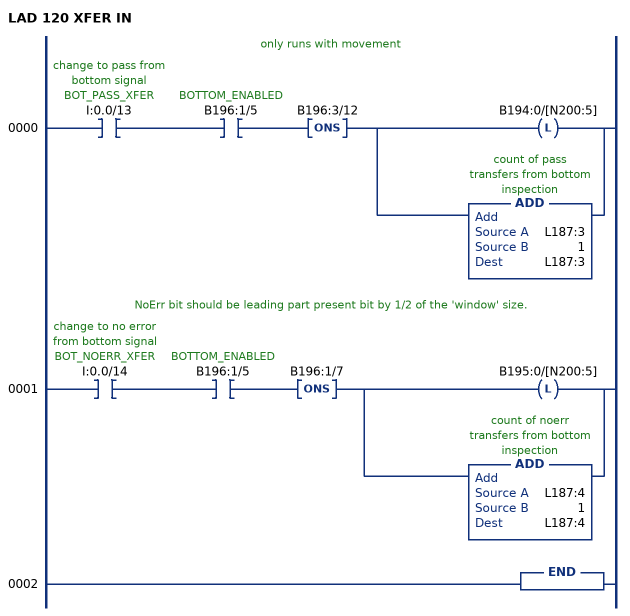
% Rung: 0 %
% only runs with movement %
SOR XIC I:0.0/13 XIC B196:1/5 ONS B196:3/12 BST OTL B194:0/[N200:5] NXB ADD L187:3 1 L187:3 BND EOR
%   I:0.0/13  BOT_PASS_XFER  "change to pass from bottom signal" %
%   B196:1/5  BOTTOM_ENABLED %
%   N200:5  TOP_LOAD %
%   L187:3  "count of pass transfers from bottom inspection" %
% Rung: 1 %
% NoErr bit should be leading part present bit by 1/2 of the 'window' size. %
SOR XIC I:0.0/14 XIC B196:1/5 ONS B196:1/7 BST OTL B195:0/[N200:5] NXB ADD L187:4 1 L187:4 BND EOR
%   I:0.0/14  BOT_NOERR_XFER  "change to no error from bottom signal" %
%   B196:1/5  BOTTOM_ENABLED %
%   N200:5  TOP_LOAD %
%   L187:4  "count of noerr transfers from bottom inspection" %
% Rung: 2 %
SOR END EOR

LADDER 121 "SIM PARTS"
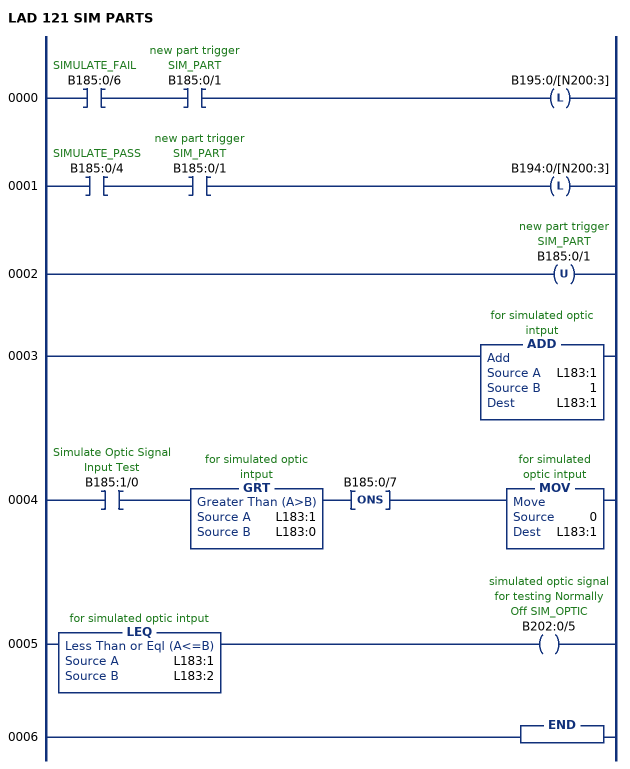
% Rung: 0 %
SOR XIC B185:0/6 XIC B185:0/1 OTL B195:0/[N200:3] EOR
%   B185:0/6  SIMULATE_FAIL %
%   B185:0/1  SIM_PART  "new part trigger" %
%   N200:3  OPT_LD_PT %
% Rung: 1 %
SOR XIC B185:0/4 XIC B185:0/1 OTL B194:0/[N200:3] EOR
%   B185:0/4  SIMULATE_PASS %
%   B185:0/1  SIM_PART  "new part trigger" %
%   N200:3  OPT_LD_PT %
% Rung: 2 %
SOR OTU B185:0/1 EOR
%   B185:0/1  SIM_PART  "new part trigger" %
% Rung: 3 %
SOR ADD L183:1 1 L183:1 EOR
%   L183:1  "for simulated optic intput" %
% Rung: 4 %
SOR XIC B185:1/0 GRT L183:1 L183:0 ONS B185:0/7 MOV 0 L183:1 EOR
%   B185:1/0  "Simulate Optic Signal Input Test" %
%   L183:1  "for simulated optic intput" %
%   L183:0  "Movement pulse count for part data injection" %
% Rung: 5 %
SOR LEQ L183:1 L183:2 OTE B202:0/5 EOR
%   L183:1  "for simulated optic intput" %
%   L183:2  "simulated part width" %
%   B202:0/5  SIM_OPTIC  "simulated optic signal for testing Normally Off" %
% Rung: 6 %
SOR END EOR

LADDER 122 "PARTDETECT"
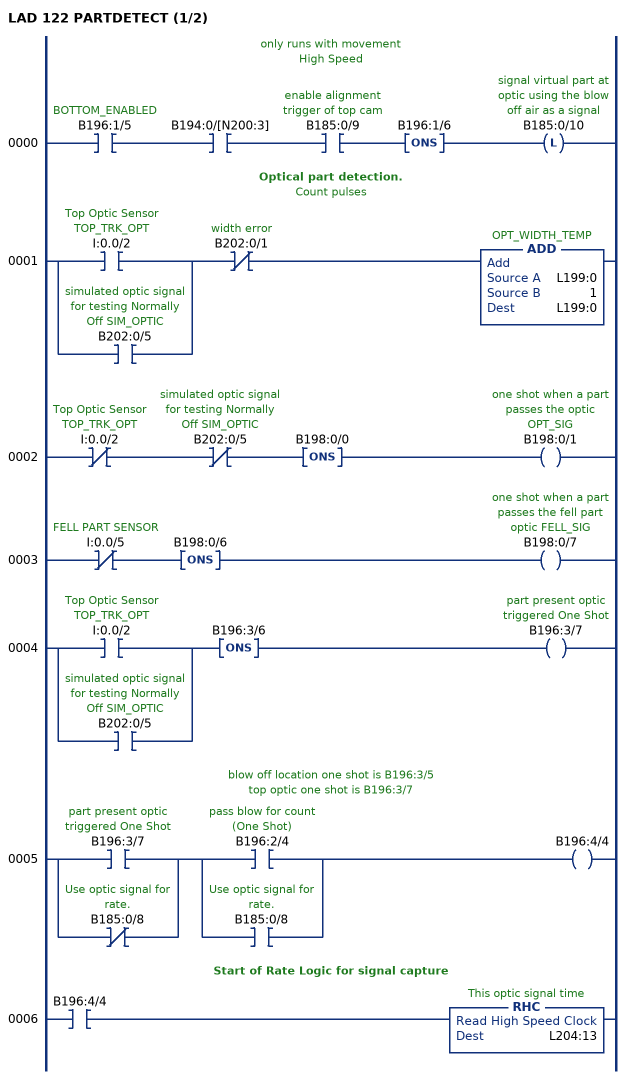
% Rung: 0 %
% only runs with movement
% High Speed %
SOR XIC B196:1/5 XIC B194:0/[N200:3] XIC B185:0/9 ONS B196:1/6 OTL B185:0/10 EOR
%   B196:1/5  BOTTOM_ENABLED %
%   N200:3  OPT_LD_PT %
%   B185:0/9  "enable alignment trigger of top cam" %
%   B185:0/10  "signal virtual part at optic using the blow off air as a signal" %
% Rung: 1 %
% TITLE: Optical part detection. %
% Count pulses %
SOR BST XIC I:0.0/2 NXB XIC B202:0/5 BND XIO B202:0/1 ADD L199:0 1 L199:0 EOR
%   I:0.0/2  TOP_TRK_OPT  "Top Optic Sensor" %
%   B202:0/5  SIM_OPTIC  "simulated optic signal for testing Normally Off" %
%   B202:0/1  "width error" %
%   L199:0  OPT_WIDTH_TEMP %
% Rung: 2 %
SOR XIO I:0.0/2 XIO B202:0/5 ONS B198:0/0 OTE B198:0/1 EOR
%   I:0.0/2  TOP_TRK_OPT  "Top Optic Sensor" %
%   B202:0/5  SIM_OPTIC  "simulated optic signal for testing Normally Off" %
%   B198:0/1  OPT_SIG  "one shot when a part passes the optic" %
% Rung: 3 %
SOR XIO I:0.0/5 ONS B198:0/6 OTE B198:0/7 EOR
%   I:0.0/5  "FELL PART SENSOR" %
%   B198:0/7  FELL_SIG  "one shot when a part passes the fell part optic" %
% Rung: 4 %
SOR BST XIC I:0.0/2 NXB XIC B202:0/5 BND ONS B196:3/6 OTE B196:3/7 EOR
%   I:0.0/2  TOP_TRK_OPT  "Top Optic Sensor" %
%   B202:0/5  SIM_OPTIC  "simulated optic signal for testing Normally Off" %
%   B196:3/7  "part present optic triggered One Shot" %
% Rung: 5 %
% blow off location one shot is B196:3/5
% top optic one shot is B196:3/7 %
SOR BST XIC B196:3/7 NXB XIO B185:0/8 BND BST XIC B196:2/4 NXB XIC B185:0/8 BND OTE B196:4/4 EOR
%   B196:3/7  "part present optic triggered One Shot" %
%   B185:0/8  "Use optic signal for rate." %
%   B196:2/4  "pass blow for count (One Shot)" %
% Rung: 6 %
% TITLE: Start of Rate Logic for signal capture %
SOR XIC B196:4/4 RHC L204:13 EOR
%   L204:13  "This optic signal time" %

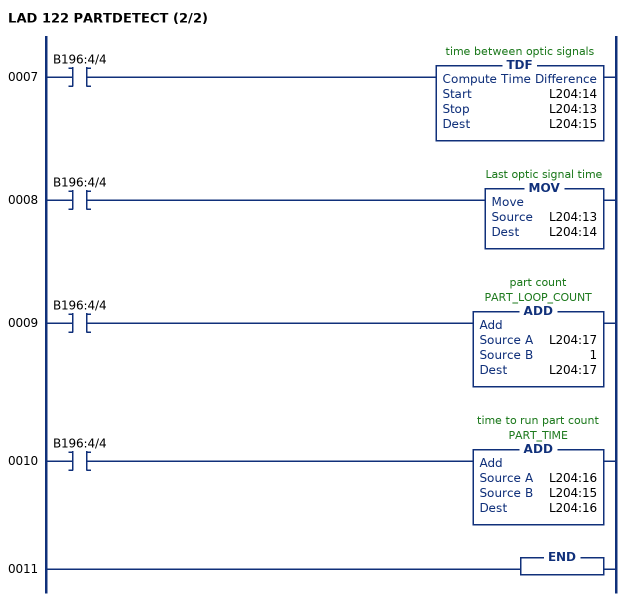
% Rung: 7 %
SOR XIC B196:4/4 TDF L204:14 L204:13 L204:15 EOR
%   L204:14  "Last optic signal time" %
%   L204:13  "This optic signal time" %
%   L204:15  "time between optic signals" %
% Rung: 8 %
SOR XIC B196:4/4 MOV L204:13 L204:14 EOR
%   L204:13  "This optic signal time" %
%   L204:14  "Last optic signal time" %
% Rung: 9 %
SOR XIC B196:4/4 ADD L204:17 1 L204:17 EOR
%   L204:17  PART_LOOP_COUNT  "part count" %
% Rung: 10 %
SOR XIC B196:4/4 ADD L204:16 L204:15 L204:16 EOR
%   L204:16  PART_TIME  "time to run part count" %
%   L204:15  "time between optic signals" %
% Rung: 11 %
SOR END EOR

LADDER 123 "OPTICWIDTH"
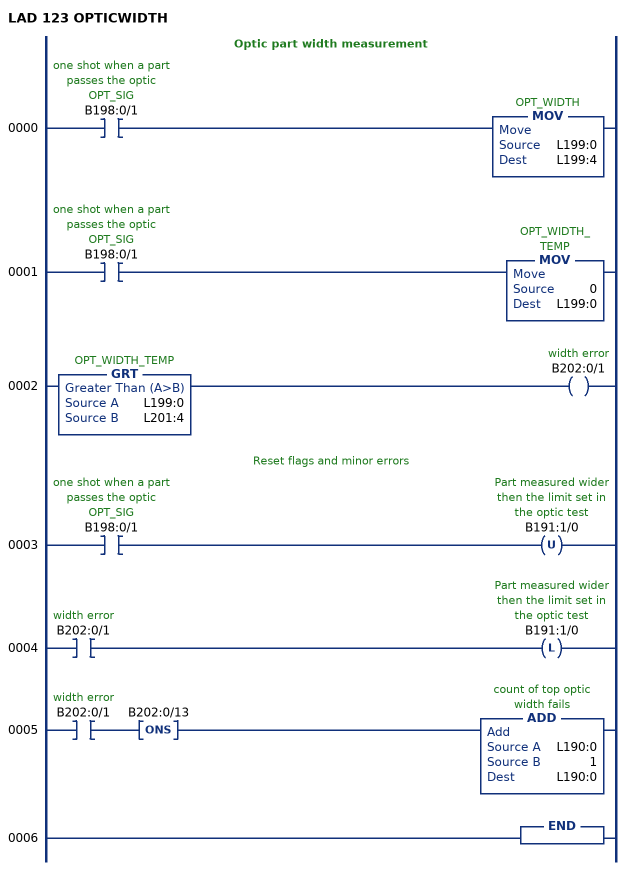
% Rung: 0 %
% TITLE: Optic part width measurement %
SOR XIC B198:0/1 MOV L199:0 L199:4 EOR
%   B198:0/1  OPT_SIG  "one shot when a part passes the optic" %
%   L199:0  OPT_WIDTH_TEMP %
%   L199:4  OPT_WIDTH %
% Rung: 1 %
SOR XIC B198:0/1 MOV 0 L199:0 EOR
%   B198:0/1  OPT_SIG  "one shot when a part passes the optic" %
%   L199:0  OPT_WIDTH_TEMP %
% Rung: 2 %
SOR GRT L199:0 L201:4 OTE B202:0/1 EOR
%   L199:0  OPT_WIDTH_TEMP %
%   L201:4  MAX_WIDTH  "hmi in" %
%   B202:0/1  "width error" %
% Rung: 3 %
% Reset flags and minor errors %
SOR XIC B198:0/1 OTU B191:1/0 EOR
%   B198:0/1  OPT_SIG  "one shot when a part passes the optic" %
%   B191:1/0  "Part measured wider then the limit set in the optic test" %
% Rung: 4 %
SOR XIC B202:0/1 OTL B191:1/0 EOR
%   B202:0/1  "width error" %
%   B191:1/0  "Part measured wider then the limit set in the optic test" %
% Rung: 5 %
SOR XIC B202:0/1 ONS B202:0/13 ADD L190:0 1 L190:0 EOR
%   B202:0/1  "width error" %
%   L190:0  "count of top optic width fails" %
% Rung: 6 %
SOR END EOR

LADDER 124 "PART GAP"
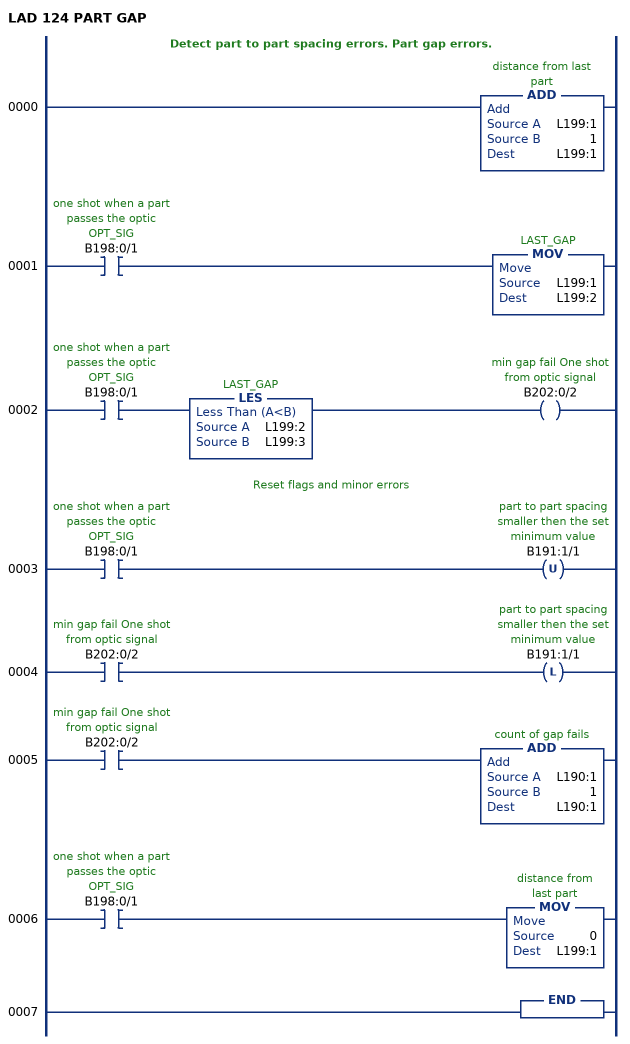
% Rung: 0 %
% TITLE: Detect part to part spacing errors. Part gap errors. %
SOR ADD L199:1 1 L199:1 EOR
%   L199:1  "distance from last part" %
% Rung: 1 %
SOR XIC B198:0/1 MOV L199:1 L199:2 EOR
%   B198:0/1  OPT_SIG  "one shot when a part passes the optic" %
%   L199:1  "distance from last part" %
%   L199:2  LAST_GAP %
% Rung: 2 %
SOR XIC B198:0/1 LES L199:2 L199:3 OTE B202:0/2 EOR
%   B198:0/1  OPT_SIG  "one shot when a part passes the optic" %
%   L199:2  LAST_GAP %
%   L199:3  MIN_WIDTH %
%   B202:0/2  "min gap fail One shot from optic signal" %
% Rung: 3 %
% Reset flags and minor errors %
SOR XIC B198:0/1 OTU B191:1/1 EOR
%   B198:0/1  OPT_SIG  "one shot when a part passes the optic" %
%   B191:1/1  "part to part spacing smaller then the set minimum value" %
% Rung: 4 %
SOR XIC B202:0/2 OTL B191:1/1 EOR
%   B202:0/2  "min gap fail One shot from optic signal" %
%   B191:1/1  "part to part spacing smaller then the set minimum value" %
% Rung: 5 %
SOR XIC B202:0/2 ADD L190:1 1 L190:1 EOR
%   B202:0/2  "min gap fail One shot from optic signal" %
%   L190:1  "count of gap fails" %
% Rung: 6 %
SOR XIC B198:0/1 MOV 0 L199:1 EOR
%   B198:0/1  OPT_SIG  "one shot when a part passes the optic" %
%   L199:1  "distance from last part" %
% Rung: 7 %
SOR END EOR

LADDER 125 "OPTIC CL"
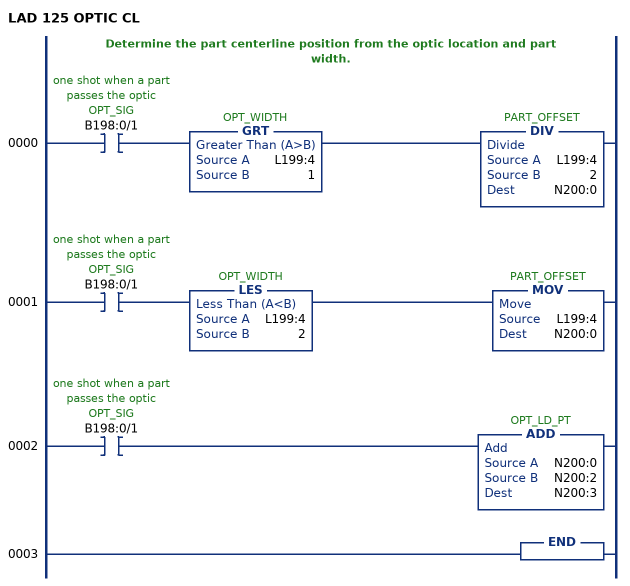
% Rung: 0 %
% TITLE: Determine the part centerline position from the optic location and part width. %
SOR XIC B198:0/1 GRT L199:4 1 DIV L199:4 2 N200:0 EOR
%   B198:0/1  OPT_SIG  "one shot when a part passes the optic" %
%   L199:4  OPT_WIDTH %
%   N200:0  PART_OFFSET %
% Rung: 1 %
SOR XIC B198:0/1 LES L199:4 2 MOV L199:4 N200:0 EOR
%   B198:0/1  OPT_SIG  "one shot when a part passes the optic" %
%   L199:4  OPT_WIDTH %
%   N200:0  PART_OFFSET %
% Rung: 2 %
SOR XIC B198:0/1 ADD N200:0 N200:2 N200:3 EOR
%   B198:0/1  OPT_SIG  "one shot when a part passes the optic" %
%   N200:0  PART_OFFSET %
%   N200:2  OPTIC_LOC %
%   N200:3  OPT_LD_PT %
% Rung: 3 %
SOR END EOR

LADDER 126 "ALIGNMENT"
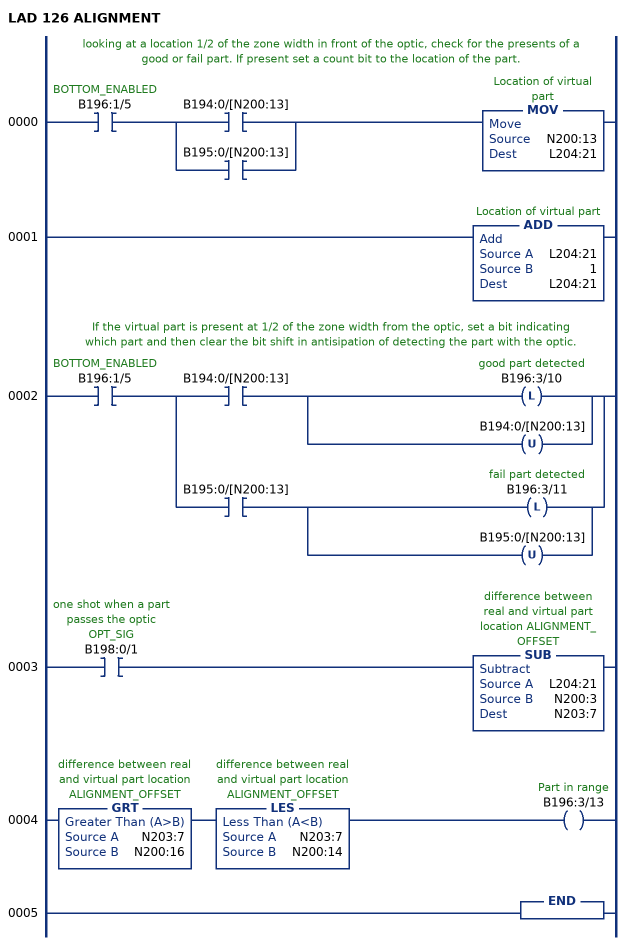
% Rung: 0 %
% looking at a location 1/2 of the zone width in front of the optic, check for the presents of a good or fail part. If present set a count bit to the location of the part. %
SOR XIC B196:1/5 BST XIC B194:0/[N200:13] NXB XIC B195:0/[N200:13] BND MOV N200:13 L204:21 EOR
%   B196:1/5  BOTTOM_ENABLED %
%   N200:13  ALIGNMENT_START_LOC %
%   L204:21  "Location of virtual part" %
% Rung: 1 %
SOR ADD L204:21 1 L204:21 EOR
%   L204:21  "Location of virtual part" %
% Rung: 2 %
% If the virtual part is present at 1/2 of the zone width from the optic, set a bit indicating which part and then clear the bit shift in antisipation of detecting the part with the optic. %
SOR XIC B196:1/5 BST XIC B194:0/[N200:13] BST OTL B196:3/10 NXB OTU B194:0/[N200:13] BND NXB XIC B195:0/[N200:13] BST OTL B196:3/11 NXB OTU B195:0/[N200:13] BND BND EOR
%   B196:1/5  BOTTOM_ENABLED %
%   N200:13  ALIGNMENT_START_LOC %
%   B196:3/10  "good part detected" %
%   B196:3/11  "fail part detected" %
% Rung: 3 %
SOR XIC B198:0/1 SUB L204:21 N200:3 N203:7 EOR
%   B198:0/1  OPT_SIG  "one shot when a part passes the optic" %
%   L204:21  "Location of virtual part" %
%   N200:3  OPT_LD_PT %
%   N203:7  ALIGNMENT_OFFSET  "difference between real and virtual part location" %
% Rung: 4 %
SOR GRT N203:7 N200:16 LES N203:7 N200:14 OTE B196:3/13 EOR
%   N203:7  ALIGNMENT_OFFSET  "difference between real and virtual part location" %
%   N200:16  "Minus one half of the transition zone" %
%   N200:14  "1/2 transistion zone" %
%   B196:3/13  "Part in range" %
% Rung: 5 %
SOR END EOR

LADDER 127 "OPTIC_LOAD"
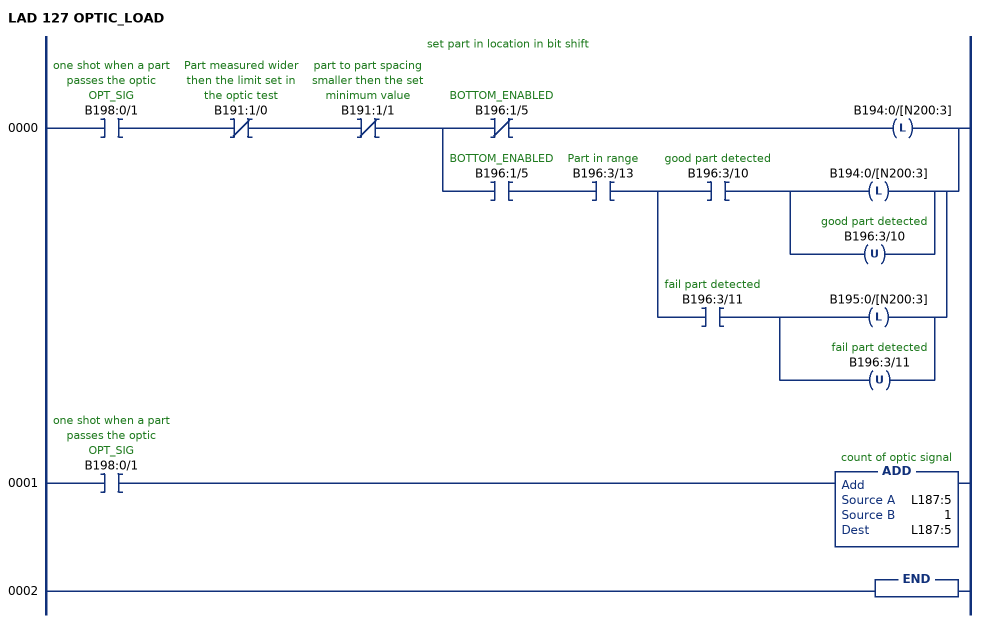
% Rung: 0 %
% set part in location in bit shift %
SOR XIC B198:0/1 XIO B191:1/0 XIO B191:1/1 BST XIO B196:1/5 OTL B194:0/[N200:3] NXB XIC B196:1/5 XIC B196:3/13 BST XIC B196:3/10 BST OTL B194:0/[N200:3] NXB OTU B196:3/10 BND NXB XIC B196:3/11 BST OTL B195:0/[N200:3] NXB OTU B196:3/11 BND BND BND EOR
%   B198:0/1  OPT_SIG  "one shot when a part passes the optic" %
%   B191:1/0  "Part measured wider then the limit set in the optic test" %
%   B191:1/1  "part to part spacing smaller then the set minimum value" %
%   B196:1/5  BOTTOM_ENABLED %
%   N200:3  OPT_LD_PT %
%   B196:3/13  "Part in range" %
%   B196:3/10  "good part detected" %
%   B196:3/11  "fail part detected" %
% Rung: 1 %
SOR XIC B198:0/1 ADD L187:5 1 L187:5 EOR
%   B198:0/1  OPT_SIG  "one shot when a part passes the optic" %
%   L187:5  "count of optic signal" %
% Rung: 2 %
SOR END EOR

LADDER 128 "FELL PART"
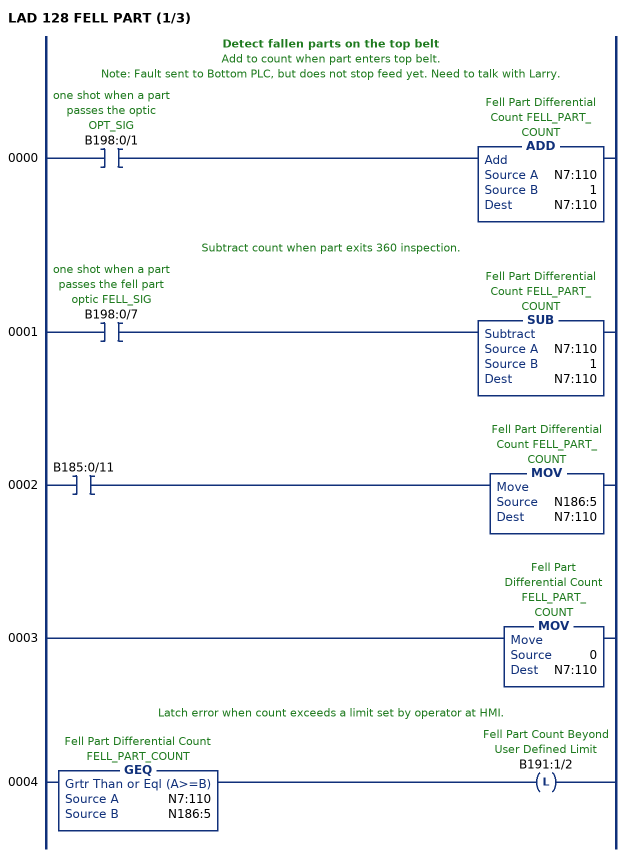
% Rung: 0 %
% TITLE: Detect fallen parts on the top belt %
% Add to count when part enters top belt.
% Note: Fault sent to Bottom PLC, but does not stop feed yet. Need to talk with Larry. %
SOR XIC B198:0/1 ADD N7:110 1 N7:110 EOR
%   B198:0/1  OPT_SIG  "one shot when a part passes the optic" %
%   N7:110  FELL_PART_COUNT  "Fell Part Differential Count" %
% Rung: 1 %
% Subtract count when part exits 360 inspection. %
SOR XIC B198:0/7 SUB N7:110 1 N7:110 EOR
%   B198:0/7  FELL_SIG  "one shot when a part passes the fell part optic" %
%   N7:110  FELL_PART_COUNT  "Fell Part Differential Count" %
% Rung: 2 %
SOR XIC B185:0/11 MOV N186:5 N7:110 EOR
%   N186:5  FELL_PART_LIMIT  "Fell Part Differential Limit From HMI" %
%   N7:110  FELL_PART_COUNT  "Fell Part Differential Count" %
% Rung: 3 %
SOR MOV 0 N7:110 EOR
%   N7:110  FELL_PART_COUNT  "Fell Part Differential Count" %
% Rung: 4 %
% Latch error when count exceeds a limit set by operator at HMI. %
SOR GEQ N7:110 N186:5 OTL B191:1/2 EOR
%   N7:110  FELL_PART_COUNT  "Fell Part Differential Count" %
%   N186:5  FELL_PART_LIMIT  "Fell Part Differential Limit From HMI" %
%   B191:1/2  "Fell Part Count Beyond User Defined Limit" %

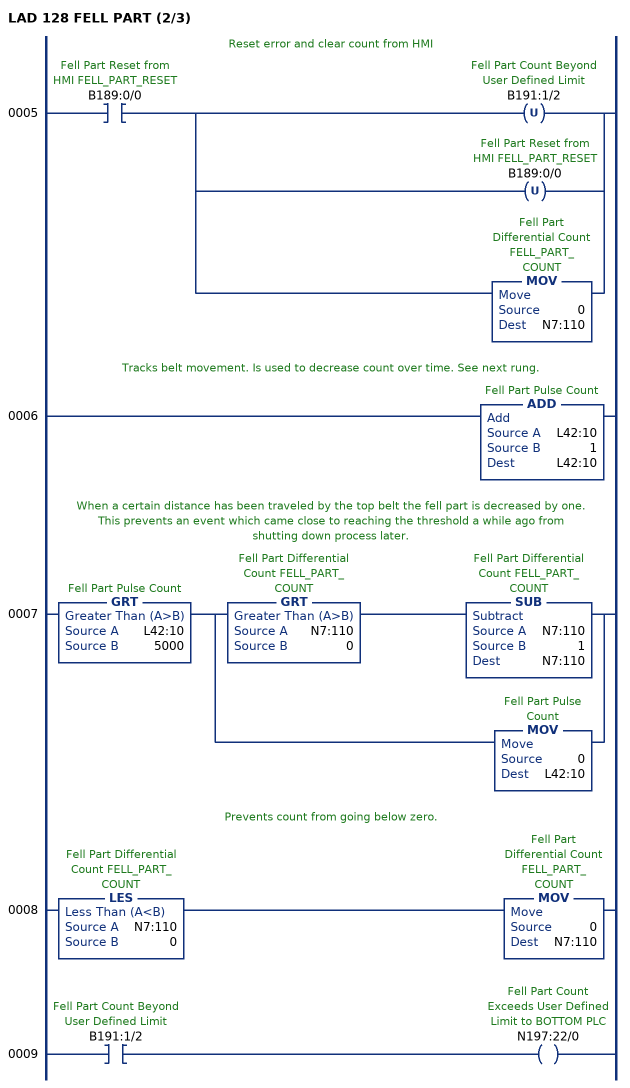
% Rung: 5 %
% Reset error and clear count from HMI %
SOR XIC B189:0/0 BST OTU B191:1/2 NXB OTU B189:0/0 NXB MOV 0 N7:110 BND EOR
%   B189:0/0  FELL_PART_RESET  "Fell Part Reset from HMI" %
%   B191:1/2  "Fell Part Count Beyond User Defined Limit" %
%   N7:110  FELL_PART_COUNT  "Fell Part Differential Count" %
% Rung: 6 %
% Tracks belt movement. Is used to decrease count over time. See next rung. %
SOR ADD L42:10 1 L42:10 EOR
%   L42:10  "Fell Part Pulse Count" %
% Rung: 7 %
% When a certain distance has been traveled by the top belt the fell part is decreased by one. This prevents an event which came close to reaching the threshold a while ago from shutting down process later. %
SOR GRT L42:10 5000 BST GRT N7:110 0 SUB N7:110 1 N7:110 NXB MOV 0 L42:10 BND EOR
%   L42:10  "Fell Part Pulse Count" %
%   N7:110  FELL_PART_COUNT  "Fell Part Differential Count" %
% Rung: 8 %
% Prevents count from going below zero. %
SOR LES N7:110 0 MOV 0 N7:110 EOR
%   N7:110  FELL_PART_COUNT  "Fell Part Differential Count" %
% Rung: 9 %
SOR XIC B191:1/2 OTE N197:22/0 EOR
%   B191:1/2  "Fell Part Count Beyond User Defined Limit" %
%   N197:22/0  "Fell Part Count Exceeds User Defined Limit to BOTTOM PLC" %

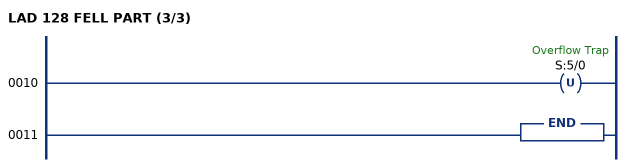
% Rung: 10 %
SOR OTU S:5/0 EOR
%   S:5/0  "Overflow Trap" %
% Rung: 11 %
SOR END EOR

LADDER 130 "INS 5 TRIG"
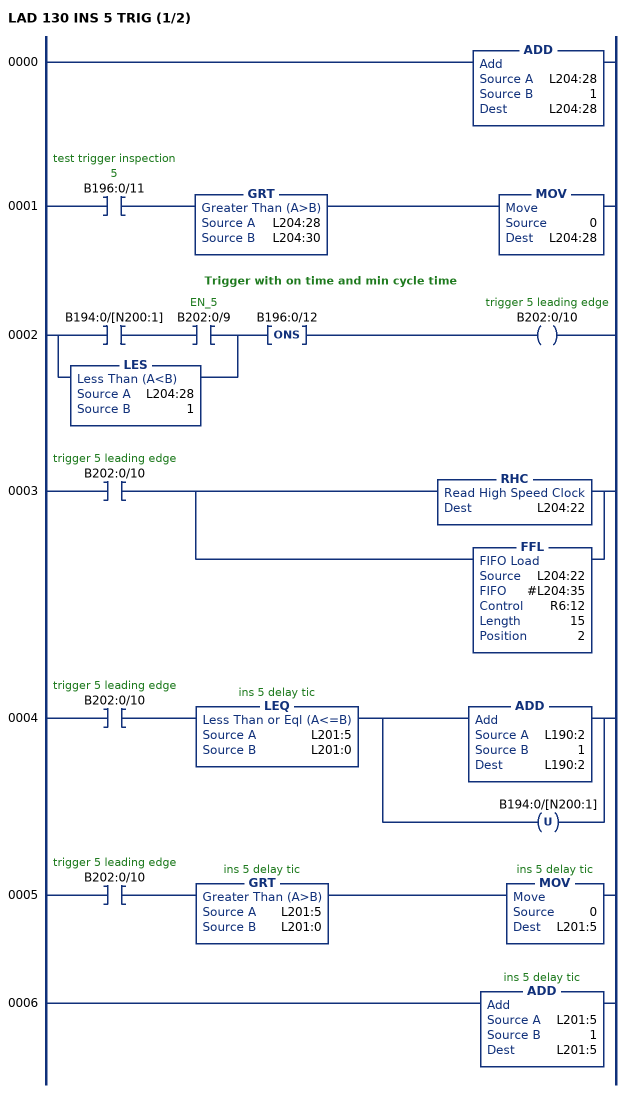
% Rung: 0 %
SOR ADD L204:28 1 L204:28 EOR
% Rung: 1 %
SOR XIC B196:0/11 GRT L204:28 L204:30 MOV 0 L204:28 EOR
%   B196:0/11  "test trigger inspection 5" %
% Rung: 2 %
% TITLE: Trigger with on time and min cycle time %
SOR BST XIC B194:0/[N200:1] XIC B202:0/9 NXB LES L204:28 1 BND ONS B196:0/12 OTE B202:0/10 EOR
%   N200:1  INS_5_TRIG_LOC %
%   B202:0/9  EN_5 %
%   B202:0/10  "trigger 5 leading edge" %
% Rung: 3 %
SOR XIC B202:0/10 BST RHC L204:22 NXB FFL L204:22 #L204:35 R6:12 15 2 BND EOR
%   B202:0/10  "trigger 5 leading edge" %
% Rung: 4 %
SOR XIC B202:0/10 LEQ L201:5 L201:0 BST ADD L190:2 1 L190:2 NXB OTU B194:0/[N200:1] BND EOR
%   B202:0/10  "trigger 5 leading edge" %
%   L201:5  "ins 5 delay tic" %
%   L201:0  CAM_5_MIN_CYCLE_TIME %
%   N200:1  INS_5_TRIG_LOC %
% Rung: 5 %
SOR XIC B202:0/10 GRT L201:5 L201:0 MOV 0 L201:5 EOR
%   B202:0/10  "trigger 5 leading edge" %
%   L201:5  "ins 5 delay tic" %
%   L201:0  CAM_5_MIN_CYCLE_TIME %
% Rung: 6 %
SOR ADD L201:5 1 L201:5 EOR
%   L201:5  "ins 5 delay tic" %

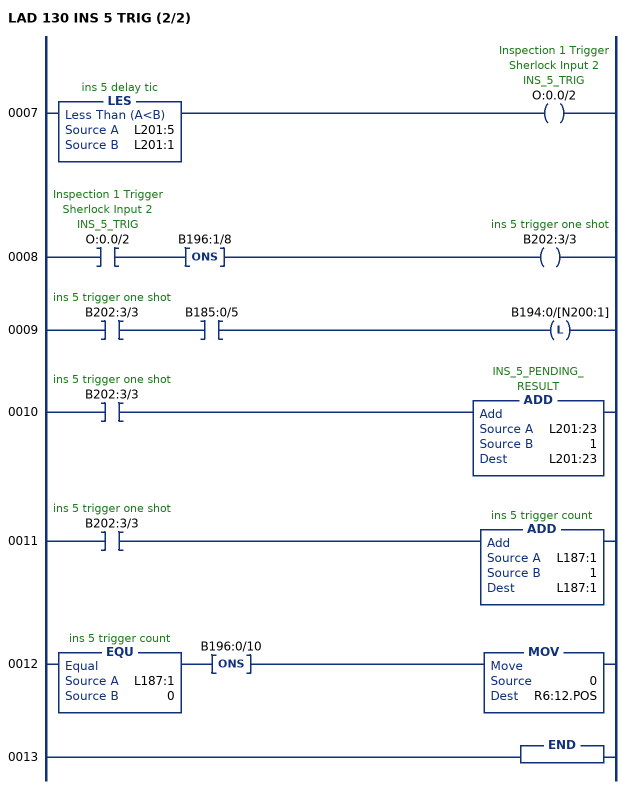
% Rung: 7 %
SOR LES L201:5 L201:1 OTE O:0.0/2 EOR
%   L201:5  "ins 5 delay tic" %
%   L201:1  CAM_5_TRIG_TIME %
%   O:0.0/2  INS_5_TRIG  "Inspection 1 Trigger Sherlock Input 2" %
% Rung: 8 %
SOR XIC O:0.0/2 ONS B196:1/8 OTE B202:3/3 EOR
%   O:0.0/2  INS_5_TRIG  "Inspection 1 Trigger Sherlock Input 2" %
%   B202:3/3  "ins 5 trigger one shot" %
% Rung: 9 %
SOR XIC B202:3/3 XIC B185:0/5 OTL B194:0/[N200:1] EOR
%   B202:3/3  "ins 5 trigger one shot" %
%   N200:1  INS_5_TRIG_LOC %
% Rung: 10 %
SOR XIC B202:3/3 ADD L201:23 1 L201:23 EOR
%   B202:3/3  "ins 5 trigger one shot" %
%   L201:23  INS_5_PENDING_RESULT %
% Rung: 11 %
SOR XIC B202:3/3 ADD L187:1 1 L187:1 EOR
%   B202:3/3  "ins 5 trigger one shot" %
%   L187:1  "ins 5 trigger count" %
% Rung: 12 %
SOR EQU L187:1 0 ONS B196:0/10 MOV 0 R6:12.POS EOR
%   L187:1  "ins 5 trigger count" %
% Rung: 13 %
SOR END EOR

LADDER 131 "INS 5 RSLT"
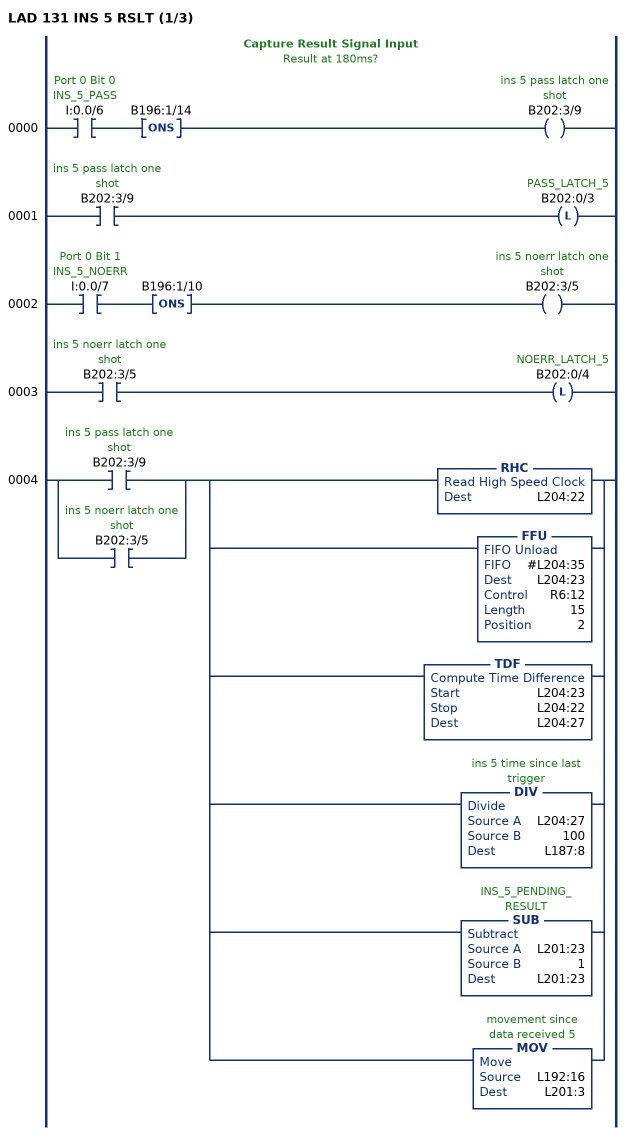
% Rung: 0 %
% TITLE: Capture Result Signal Input %
% Result at 180ms? %
SOR XIC I:0.0/6 ONS B196:1/14 OTE B202:3/9 EOR
%   I:0.0/6  INS_5_PASS  "Port 0 Bit 0" %
%   B202:3/9  "ins 5 pass latch one shot" %
% Rung: 1 %
SOR XIC B202:3/9 OTL B202:0/3 EOR
%   B202:3/9  "ins 5 pass latch one shot" %
%   B202:0/3  PASS_LATCH_5 %
% Rung: 2 %
SOR XIC I:0.0/7 ONS B196:1/10 OTE B202:3/5 EOR
%   I:0.0/7  INS_5_NOERR  "Port 0 Bit 1" %
%   B202:3/5  "ins 5 noerr latch one shot" %
% Rung: 3 %
SOR XIC B202:3/5 OTL B202:0/4 EOR
%   B202:3/5  "ins 5 noerr latch one shot" %
%   B202:0/4  NOERR_LATCH_5 %
% Rung: 4 %
SOR BST XIC B202:3/9 NXB XIC B202:3/5 BND BST RHC L204:22 NXB FFU #L204:35 L204:23 R6:12 15 2 NXB TDF L204:23 L204:22 L204:27 NXB DIV L204:27 100 L187:8 NXB SUB L201:23 1 L201:23 NXB MOV L192:16 L201:3 BND EOR
%   B202:3/9  "ins 5 pass latch one shot" %
%   B202:3/5  "ins 5 noerr latch one shot" %
%   L187:8  "ins 5 time since last trigger" %
%   L201:23  INS_5_PENDING_RESULT %
%   L192:16  COMBINED_OFFSET  "use this offset value for looking for the part present bit after an inspeciton" %
%   L201:3  "movement since data received 5" %

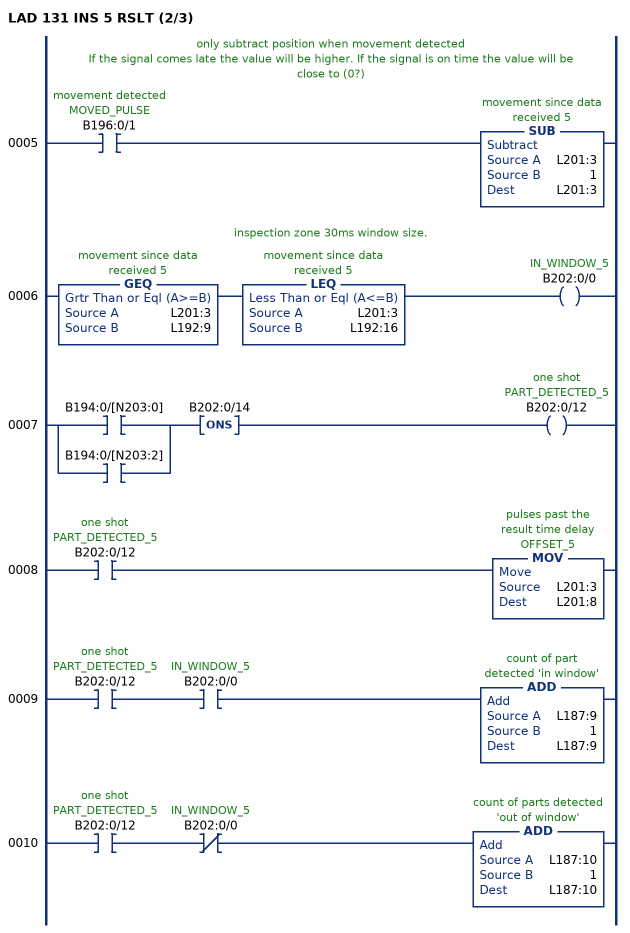
% Rung: 5 %
% only subtract position when movement detected
% If the signal comes late the value will be higher. If the signal is on time the value will be close to (0?) %
SOR XIC B196:0/1 SUB L201:3 1 L201:3 EOR
%   B196:0/1  MOVED_PULSE  "movement detected" %
%   L201:3  "movement since data received 5" %
% Rung: 6 %
% inspection zone 30ms window size. %
SOR GEQ L201:3 L192:9 LEQ L201:3 L192:16 OTE B202:0/0 EOR
%   L201:3  "movement since data received 5" %
%   L192:9  RESULT_OFFSET  "in pulses" %
%   L192:16  COMBINED_OFFSET  "use this offset value for looking for the part present bit after an inspeciton" %
%   B202:0/0  IN_WINDOW_5 %
% Rung: 7 %
SOR BST XIC B194:0/[N203:0] NXB XIC B194:0/[N203:2] BND ONS B202:0/14 OTE B202:0/12 EOR
%   N203:0  INS_5_TEST_LOC1  "result + offset shift" %
%   N203:2  INS_5_TEST_LOC2 %
%   B202:0/12  PART_DETECTED_5  "one shot" %
% Rung: 8 %
SOR XIC B202:0/12 MOV L201:3 L201:8 EOR
%   B202:0/12  PART_DETECTED_5  "one shot" %
%   L201:3  "movement since data received 5" %
%   L201:8  OFFSET_5  "pulses past the result time delay" %
% Rung: 9 %
SOR XIC B202:0/12 XIC B202:0/0 ADD L187:9 1 L187:9 EOR
%   B202:0/12  PART_DETECTED_5  "one shot" %
%   B202:0/0  IN_WINDOW_5 %
%   L187:9  "count of part detected 'in window'" %
% Rung: 10 %
SOR XIC B202:0/12 XIO B202:0/0 ADD L187:10 1 L187:10 EOR
%   B202:0/12  PART_DETECTED_5  "one shot" %
%   B202:0/0  IN_WINDOW_5 %
%   L187:10  "count of parts detected 'out of window'" %

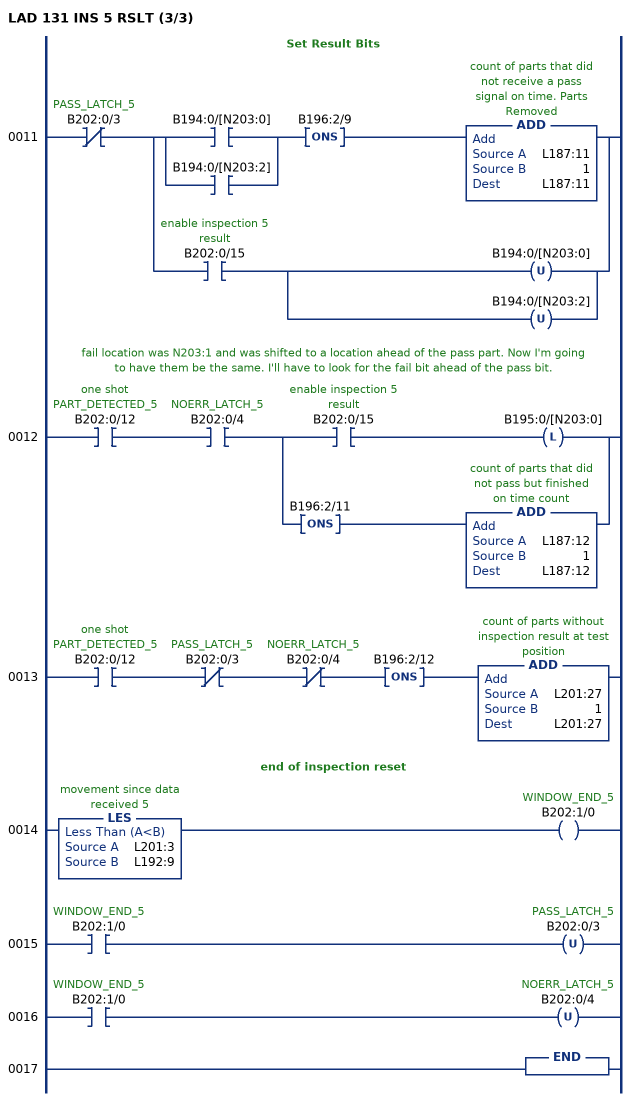
% Rung: 11 %
% TITLE: Set Result Bits %
SOR XIO B202:0/3 BST BST XIC B194:0/[N203:0] NXB XIC B194:0/[N203:2] BND ONS B196:2/9 ADD L187:11 1 L187:11 NXB XIC B202:0/15 BST OTU B194:0/[N203:0] NXB OTU B194:0/[N203:2] BND BND EOR
%   B202:0/3  PASS_LATCH_5 %
%   N203:0  INS_5_TEST_LOC1  "result + offset shift" %
%   N203:2  INS_5_TEST_LOC2 %
%   L187:11  "count of parts that did not receive a pass signal on time. Parts Removed" %
%   B202:0/15  "enable inspection 5 result" %
% Rung: 12 %
% fail location was N203:1 and was shifted to a location ahead of the pass part. Now I'm going to have them be the same. I'll have to look for the fail bit ahead of the pass bit. %
SOR XIC B202:0/12 XIC B202:0/4 BST XIC B202:0/15 OTL B195:0/[N203:0] NXB ONS B196:2/11 ADD L187:12 1 L187:12 BND EOR
%   B202:0/12  PART_DETECTED_5  "one shot" %
%   B202:0/4  NOERR_LATCH_5 %
%   B202:0/15  "enable inspection 5 result" %
%   N203:0  INS_5_TEST_LOC1  "result + offset shift" %
%   L187:12  "count of parts that did not pass but finished on time count" %
% Rung: 13 %
SOR XIC B202:0/12 XIO B202:0/3 XIO B202:0/4 ONS B196:2/12 ADD L201:27 1 L201:27 EOR
%   B202:0/12  PART_DETECTED_5  "one shot" %
%   B202:0/3  PASS_LATCH_5 %
%   B202:0/4  NOERR_LATCH_5 %
%   L201:27  "count of parts without inspection result at test position" %
% Rung: 14 %
% TITLE: end of inspection reset %
SOR LES L201:3 L192:9 OTE B202:1/0 EOR
%   L201:3  "movement since data received 5" %
%   L192:9  RESULT_OFFSET  "in pulses" %
%   B202:1/0  WINDOW_END_5 %
% Rung: 15 %
SOR XIC B202:1/0 OTU B202:0/3 EOR
%   B202:1/0  WINDOW_END_5 %
%   B202:0/3  PASS_LATCH_5 %
% Rung: 16 %
SOR XIC B202:1/0 OTU B202:0/4 EOR
%   B202:1/0  WINDOW_END_5 %
%   B202:0/4  NOERR_LATCH_5 %
% Rung: 17 %
SOR END EOR

LADDER 140 "INS 6 TRIG"
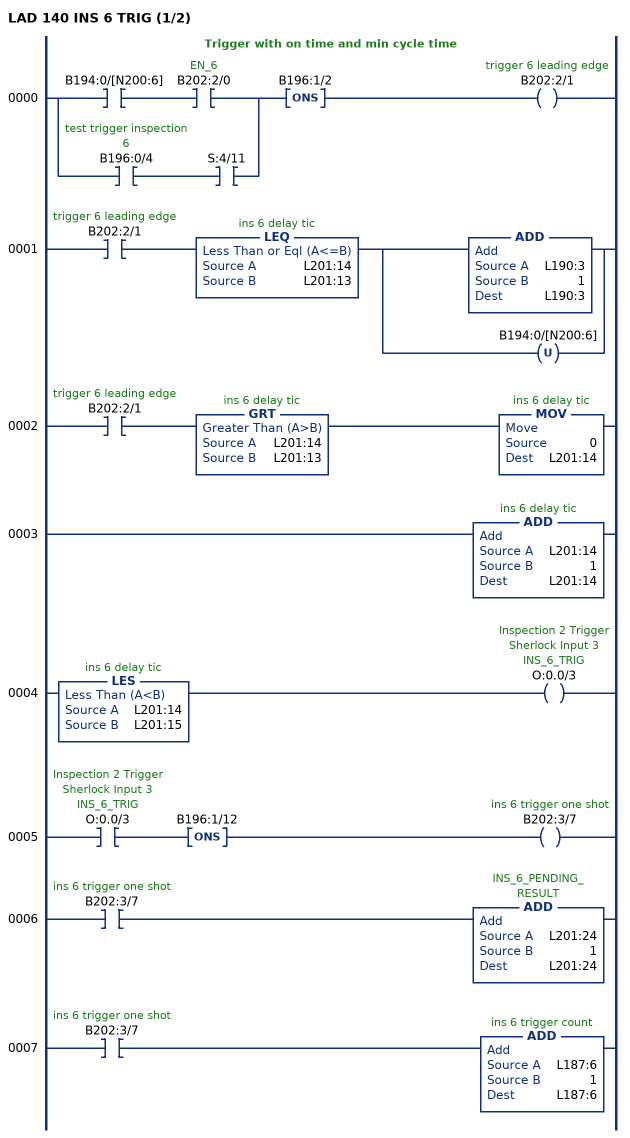
% Rung: 0 %
% TITLE: Trigger with on time and min cycle time %
SOR BST XIC B194:0/[N200:6] XIC B202:2/0 NXB XIC B196:0/4 XIC S:4/11 BND ONS B196:1/2 OTE B202:2/1 EOR
%   N200:6  INS_6_TRIG_LOC %
%   B202:2/0  EN_6 %
%   B196:0/4  "test trigger inspection 6" %
%   B202:2/1  "trigger 6 leading edge" %
% Rung: 1 %
SOR XIC B202:2/1 LEQ L201:14 L201:13 BST ADD L190:3 1 L190:3 NXB OTU B194:0/[N200:6] BND EOR
%   B202:2/1  "trigger 6 leading edge" %
%   L201:14  "ins 6 delay tic" %
%   L201:13  CAM_6_MIN_CYCLE_TIME %
%   N200:6  INS_6_TRIG_LOC %
% Rung: 2 %
SOR XIC B202:2/1 GRT L201:14 L201:13 MOV 0 L201:14 EOR
%   B202:2/1  "trigger 6 leading edge" %
%   L201:14  "ins 6 delay tic" %
%   L201:13  CAM_6_MIN_CYCLE_TIME %
% Rung: 3 %
SOR ADD L201:14 1 L201:14 EOR
%   L201:14  "ins 6 delay tic" %
% Rung: 4 %
SOR LES L201:14 L201:15 OTE O:0.0/3 EOR
%   L201:14  "ins 6 delay tic" %
%   L201:15  CAM_6_TRIG_TIME %
%   O:0.0/3  INS_6_TRIG  "Inspection 2 Trigger Sherlock Input 3" %
% Rung: 5 %
SOR XIC O:0.0/3 ONS B196:1/12 OTE B202:3/7 EOR
%   O:0.0/3  INS_6_TRIG  "Inspection 2 Trigger Sherlock Input 3" %
%   B202:3/7  "ins 6 trigger one shot" %
% Rung: 6 %
SOR XIC B202:3/7 ADD L201:24 1 L201:24 EOR
%   B202:3/7  "ins 6 trigger one shot" %
%   L201:24  INS_6_PENDING_RESULT %
% Rung: 7 %
SOR XIC B202:3/7 ADD L187:6 1 L187:6 EOR
%   B202:3/7  "ins 6 trigger one shot" %
%   L187:6  "ins 6 trigger count" %

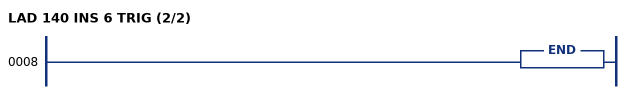
% Rung: 8 %
SOR END EOR

LADDER 141 "INS 6 RSLT"
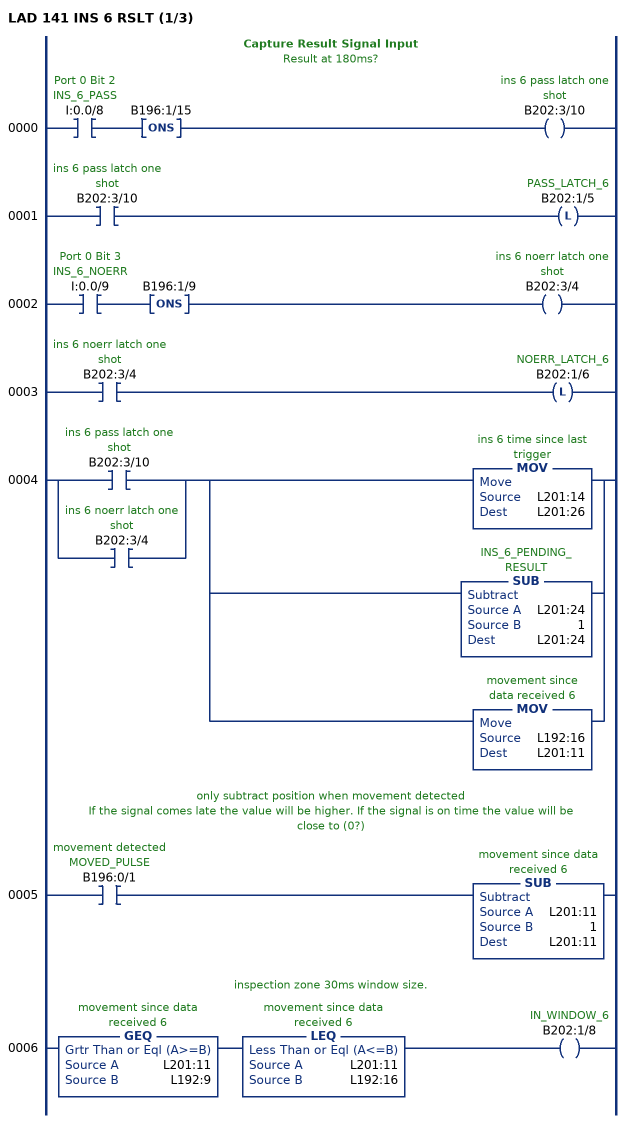
% Rung: 0 %
% TITLE: Capture Result Signal Input %
% Result at 180ms? %
SOR XIC I:0.0/8 ONS B196:1/15 OTE B202:3/10 EOR
%   I:0.0/8  INS_6_PASS  "Port 0 Bit 2" %
%   B202:3/10  "ins 6 pass latch one shot" %
% Rung: 1 %
SOR XIC B202:3/10 OTL B202:1/5 EOR
%   B202:3/10  "ins 6 pass latch one shot" %
%   B202:1/5  PASS_LATCH_6 %
% Rung: 2 %
SOR XIC I:0.0/9 ONS B196:1/9 OTE B202:3/4 EOR
%   I:0.0/9  INS_6_NOERR  "Port 0 Bit 3" %
%   B202:3/4  "ins 6 noerr latch one shot" %
% Rung: 3 %
SOR XIC B202:3/4 OTL B202:1/6 EOR
%   B202:3/4  "ins 6 noerr latch one shot" %
%   B202:1/6  NOERR_LATCH_6 %
% Rung: 4 %
SOR BST XIC B202:3/10 NXB XIC B202:3/4 BND BST MOV L201:14 L201:26 NXB SUB L201:24 1 L201:24 NXB MOV L192:16 L201:11 BND EOR
%   B202:3/10  "ins 6 pass latch one shot" %
%   B202:3/4  "ins 6 noerr latch one shot" %
%   L201:14  "ins 6 delay tic" %
%   L201:26  "ins 6 time since last trigger" %
%   L201:24  INS_6_PENDING_RESULT %
%   L192:16  COMBINED_OFFSET  "use this offset value for looking for the part present bit after an inspeciton" %
%   L201:11  "movement since data received 6" %
% Rung: 5 %
% only subtract position when movement detected
% If the signal comes late the value will be higher. If the signal is on time the value will be close to (0?) %
SOR XIC B196:0/1 SUB L201:11 1 L201:11 EOR
%   B196:0/1  MOVED_PULSE  "movement detected" %
%   L201:11  "movement since data received 6" %
% Rung: 6 %
% inspection zone 30ms window size. %
SOR GEQ L201:11 L192:9 LEQ L201:11 L192:16 OTE B202:1/8 EOR
%   L201:11  "movement since data received 6" %
%   L192:9  RESULT_OFFSET  "in pulses" %
%   L192:16  COMBINED_OFFSET  "use this offset value for looking for the part present bit after an inspeciton" %
%   B202:1/8  IN_WINDOW_6 %

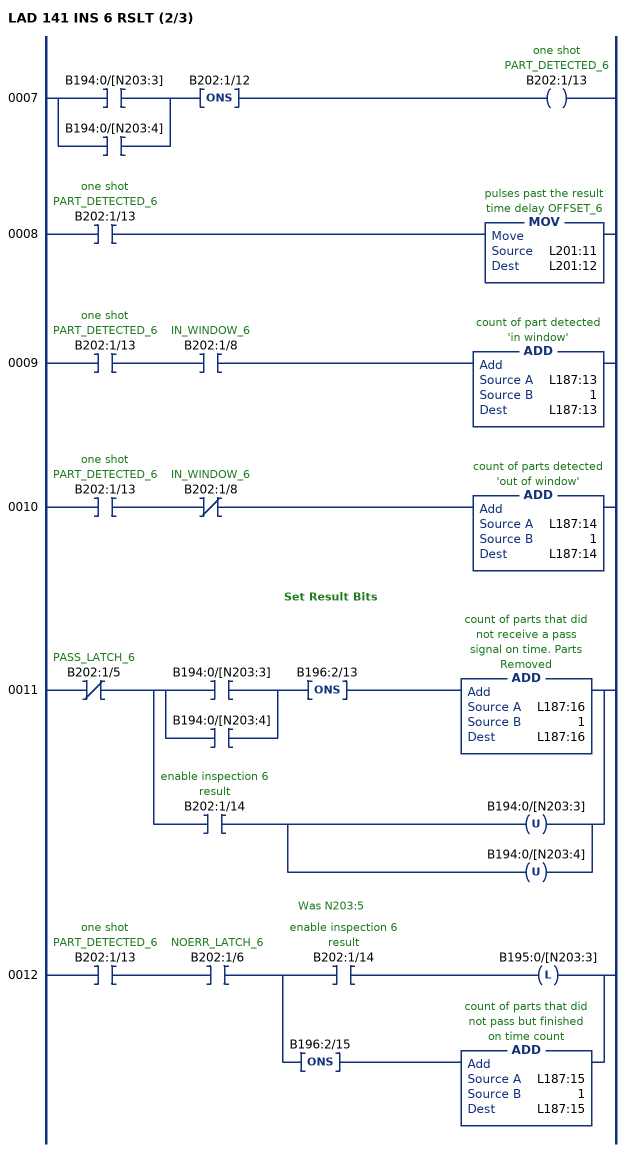
% Rung: 7 %
SOR BST XIC B194:0/[N203:3] NXB XIC B194:0/[N203:4] BND ONS B202:1/12 OTE B202:1/13 EOR
%   N203:3  INS_6_TEST_LOC1  "result + offset shift" %
%   N203:4  INS_6_TEST_LOC2 %
%   B202:1/13  PART_DETECTED_6  "one shot" %
% Rung: 8 %
SOR XIC B202:1/13 MOV L201:11 L201:12 EOR
%   B202:1/13  PART_DETECTED_6  "one shot" %
%   L201:11  "movement since data received 6" %
%   L201:12  OFFSET_6  "pulses past the result time delay" %
% Rung: 9 %
SOR XIC B202:1/13 XIC B202:1/8 ADD L187:13 1 L187:13 EOR
%   B202:1/13  PART_DETECTED_6  "one shot" %
%   B202:1/8  IN_WINDOW_6 %
%   L187:13  "count of part detected 'in window'" %
% Rung: 10 %
SOR XIC B202:1/13 XIO B202:1/8 ADD L187:14 1 L187:14 EOR
%   B202:1/13  PART_DETECTED_6  "one shot" %
%   B202:1/8  IN_WINDOW_6 %
%   L187:14  "count of parts detected 'out of window'" %
% Rung: 11 %
% TITLE: Set Result Bits %
SOR XIO B202:1/5 BST BST XIC B194:0/[N203:3] NXB XIC B194:0/[N203:4] BND ONS B196:2/13 ADD L187:16 1 L187:16 NXB XIC B202:1/14 BST OTU B194:0/[N203:3] NXB OTU B194:0/[N203:4] BND BND EOR
%   B202:1/5  PASS_LATCH_6 %
%   N203:3  INS_6_TEST_LOC1  "result + offset shift" %
%   N203:4  INS_6_TEST_LOC2 %
%   L187:16  "count of parts that did not receive a pass signal on time. Parts Removed" %
%   B202:1/14  "enable inspection 6 result" %
% Rung: 12 %
% Was N203:5 %
SOR XIC B202:1/13 XIC B202:1/6 BST XIC B202:1/14 OTL B195:0/[N203:3] NXB ONS B196:2/15 ADD L187:15 1 L187:15 BND EOR
%   B202:1/13  PART_DETECTED_6  "one shot" %
%   B202:1/6  NOERR_LATCH_6 %
%   B202:1/14  "enable inspection 6 result" %
%   N203:3  INS_6_TEST_LOC1  "result + offset shift" %
%   L187:15  "count of parts that did not pass but finished on time count" %

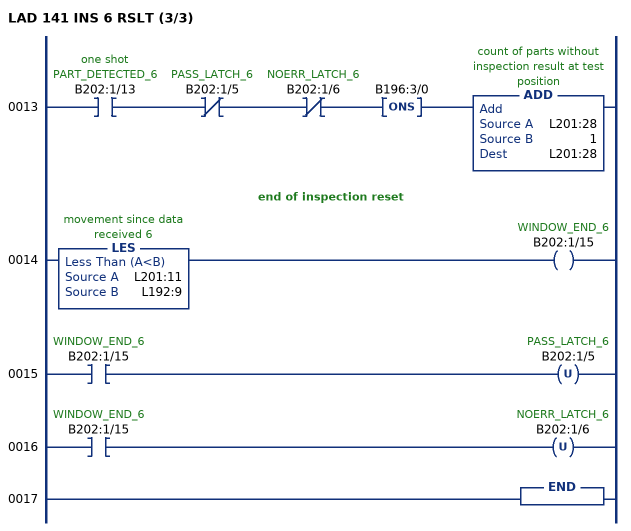
% Rung: 13 %
SOR XIC B202:1/13 XIO B202:1/5 XIO B202:1/6 ONS B196:3/0 ADD L201:28 1 L201:28 EOR
%   B202:1/13  PART_DETECTED_6  "one shot" %
%   B202:1/5  PASS_LATCH_6 %
%   B202:1/6  NOERR_LATCH_6 %
%   L201:28  "count of parts without inspection result at test position" %
% Rung: 14 %
% TITLE: end of inspection reset %
SOR LES L201:11 L192:9 OTE B202:1/15 EOR
%   L201:11  "movement since data received 6" %
%   L192:9  RESULT_OFFSET  "in pulses" %
%   B202:1/15  WINDOW_END_6 %
% Rung: 15 %
SOR XIC B202:1/15 OTU B202:1/5 EOR
%   B202:1/15  WINDOW_END_6 %
%   B202:1/5  PASS_LATCH_6 %
% Rung: 16 %
SOR XIC B202:1/15 OTU B202:1/6 EOR
%   B202:1/15  WINDOW_END_6 %
%   B202:1/6  NOERR_LATCH_6 %
% Rung: 17 %
SOR END EOR

LADDER 150 "INS 7 TRIG"
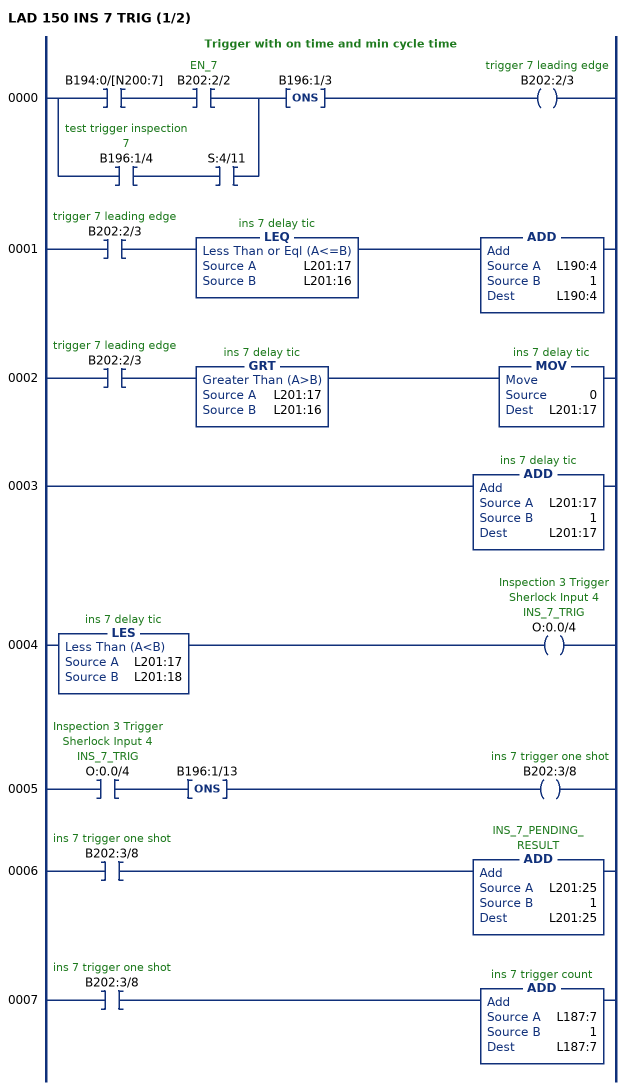
% Rung: 0 %
% TITLE: Trigger with on time and min cycle time %
SOR BST XIC B194:0/[N200:7] XIC B202:2/2 NXB XIC B196:1/4 XIC S:4/11 BND ONS B196:1/3 OTE B202:2/3 EOR
%   N200:7  INS_7_TRIG_LOC %
%   B202:2/2  EN_7 %
%   B196:1/4  "test trigger inspection 7" %
%   B202:2/3  "trigger 7 leading edge" %
% Rung: 1 %
SOR XIC B202:2/3 LEQ L201:17 L201:16 ADD L190:4 1 L190:4 EOR
%   B202:2/3  "trigger 7 leading edge" %
%   L201:17  "ins 7 delay tic" %
%   L201:16  CAM_7_MIN_CYCLE_TIME %
% Rung: 2 %
SOR XIC B202:2/3 GRT L201:17 L201:16 MOV 0 L201:17 EOR
%   B202:2/3  "trigger 7 leading edge" %
%   L201:17  "ins 7 delay tic" %
%   L201:16  CAM_7_MIN_CYCLE_TIME %
% Rung: 3 %
SOR ADD L201:17 1 L201:17 EOR
%   L201:17  "ins 7 delay tic" %
% Rung: 4 %
SOR LES L201:17 L201:18 OTE O:0.0/4 EOR
%   L201:17  "ins 7 delay tic" %
%   L201:18  CAM_7_TRIG_TIME %
%   O:0.0/4  INS_7_TRIG  "Inspection 3 Trigger Sherlock Input 4" %
% Rung: 5 %
SOR XIC O:0.0/4 ONS B196:1/13 OTE B202:3/8 EOR
%   O:0.0/4  INS_7_TRIG  "Inspection 3 Trigger Sherlock Input 4" %
%   B202:3/8  "ins 7 trigger one shot" %
% Rung: 6 %
SOR XIC B202:3/8 ADD L201:25 1 L201:25 EOR
%   B202:3/8  "ins 7 trigger one shot" %
%   L201:25  INS_7_PENDING_RESULT %
% Rung: 7 %
SOR XIC B202:3/8 ADD L187:7 1 L187:7 EOR
%   B202:3/8  "ins 7 trigger one shot" %
%   L187:7  "ins 7 trigger count" %

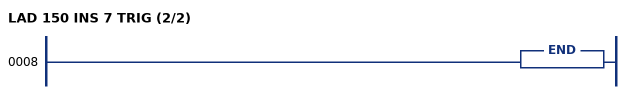
% Rung: 8 %
SOR END EOR

LADDER 151 "INS 7 RSLT"
